// TwinCAT 3 PLC project Untitled1
// ProgramVersion: 3.1.4023.0
// libraries:
//   Tc2_Standard, * (Beckhoff Automation GmbH)
//   Tc2_System, * (Beckhoff Automation GmbH)
//   Tc2_TcpIp, * (Beckhoff Automation GmbH)
//   Tc3_Module, * (Beckhoff Automation GmbH)
//   Tc2_Utilities,3.3.47.0,Beckhoff Automation GmbH
//   VisuSymbols,3.5.10.0,System
// project tree:
//   / GlobalTextList.TcGTLO, PlcTask.TcTTO, Visualization Manager.TcVMO (not stored)
//   GVLs/ GVL.TcGVL
//   POUs/ MAIN.TcPOU
//   VISUs/ Visualization.TcVIS
// real-time tasks:
//   TASK PlcTask: cycle T#10ms, priority 20, ADS port 350

CONFIGURATION Untitled1
    RESOURCE PLC ON TwinCAT3
        TASK PlcTask(INTERVAL := T#10ms, PRIORITY := 20);
        PROGRAM MAIN WITH PlcTask : MAIN;
    END_RESOURCE
END_CONFIGURATION

// ---- GVLs/GVL.TcGVL
{attribute 'qualified_only'}
VAR_GLOBAL
	
	g_bStart    AT %I* : BOOL;
	g_nConnected : INT;
	g_sWinner : STRING;
	
	g_nShake1      : INT;
	g_nShake2    : INT;
	g_nShakeWin 				:INT := 500;
END_VAR

// ---- POUs/MAIN.TcPOU
PROGRAM MAIN
VAR
	fbUdpCreate 			: FB_SocketUdpCreate;
	fbUdpCreate2 			: FB_SocketUdpCreate;
	fbSocketSend  			: FB_SocketUdpSendTo;
	fbSocketReceive 		: FB_SocketUdpReceiveFrom;
	fbSocketSend2  			: FB_SocketUdpSendTo;
	fbSocketReceive2 		: FB_SocketUdpReceiveFrom;
	fbSocketClose			: FB_SocketClose;
	fbCloseAll				: FB_SocketCloseAll;	

	sLocalHost				: T_IPv4Addr 	:= '192.168.0.253';(* Local address: String containing an (Ipv4) Internet Protocol dotted address. *)
	nLocalPort				: UDINT			:= 24042;(* Local address: IP port number. *)
	nLocalPort2				: UDINT			:= 24043;(* Local address: IP port number. *)
	sRemoteHost				: T_IPv4Addr;// 	:= '192.168.0.101';(* Remote address: String containing an (Ipv4) Internet Protocol dotted address. *)
	nRemotePort				: UDINT 	;//	:= 62510;(* Remote address: IP port number. *)
	sRemoteHost2			: T_IPv4Addr;	(* Remote address: String containing an (Ipv4) Internet Protocol dotted address. *)
	nRemotePort2			: UDINT 	;   (* Remote address: IP port number. *)
	
	sOK						: STRING		:= 'B';
	sWIN					: STRING		:= 'W';
	sLOSE					: STRING		:= 'L';
	sNumberReceive			: STRING    	:= '';
	sNumberReceive2			: STRING    	:= '';
	sStartSignal			: STRING   		:= 'A';
	sStart					: STRING 		:= 'S';
	bInitialize				: BOOL := TRUE;
	bUdpCreated				: BOOL;
	bUdpCreated2			: BOOL;
	nState 					: INT;
	bEnable 				: BOOL 	:= TRUE;
	nErrorId    : UDINT;
	fbCreateTimer	: TON := ( PT := T#100MS);

	bVar					: BOOL;
	
	nShake1 				:INT := 0;
	nShake2 				:INT := 0;
	nNumber 				:INT := 0;
	pCurrentSocket 			:T_HSOCKET;
	hSocket: INT;
	nsh: BOOL;
END_VAR

fbCloseAll( bExecute:= bInitialize);
IF fbCloseAll.bBusy OR fbCloseAll.bError THEN
	nErrorId := fbCloseAll.nErrId;
	RETURN;
END_IF
bInitialize := FALSE;

//fbUdpCreate(nLocalPort := nLocalPort, sLocalHost := sLocalHost, bExecute := TRUE );

//fbSocketSend(nRemotePort := nRemotePort,  sRemoteHost := sRemoteHost, hSocket := fbUdpCreate.hSocket, cbLen := SIZEOF(nNumber), pSrc := ADR(nNumber), bExecute := TRUE);


CASE nState OF
0:
	IF bEnable THEN
		bUdpCreated := FALSE;
		nState := 1;
	END_IF
1:
	fbUdpCreate( bExecute := FALSE );
	fbUdpCreate2( bExecute := FALSE );
	fbUdpCreate( nLocalPort := nLocalPort, sLocalHost := sLocalHost, bExecute := TRUE );
	fbUdpCreate2( nLocalPort := nLocalPort2, sLocalHost := sLocalHost, bExecute := TRUE );
	nState := 2;
2:
	fbUdpCreate( bExecute:=FALSE );
	fbUdpCreate2( bExecute:=FALSE );
	IF NOT (fbUdpCreate.bBusy AND fbUdpCreate2.bBusy) THEN
		IF NOT (fbUdpCreate.bError AND fbUdpCreate2.bError) THEN
			bUdpCreated := TRUE;
			bUdpCreated2 := TRUE;
			//fbSocketReceive( bExecute := FALSE );
			
			fbSocketReceive( hSocket := fbUdpCreate.hSocket, cbLen := 1, pDest := ADR(sNumberReceive), bExecute := TRUE , tTimeout := T#100S);
			
			
			nState := 3;
		ELSE
			nState := 100;
		END_IF
	END_IF
3:

	fbSocketReceive( bExecute := FALSE );
		IF NOT fbSocketReceive.bBusy THEN
			IF NOT fbSocketReceive.bError THEN
				//nStringInt := StringToInt(in := sNumberReceive);
				IF (bVar := sNumberReceive <> 'A') THEN
					nState := 11;
				ELSE
					sRemoteHost := fbSocketReceive.sRemoteHost;
					nRemotePort := fbSocketReceive.nRemotePort;
					nState := 23;
					GVL.g_nConnected := 1;
					fbSocketReceive2( hSocket := fbUdpCreate2.hSocket, cbLen := 1, pDest := ADR(sNumberReceive2), bExecute := TRUE , tTimeout := T#100S);
				END_IF
				
			ELSE
				nState := 100;
			END_IF
		END_IF
23:
	fbSocketReceive2( bExecute := FALSE );
		IF NOT fbSocketReceive2.bBusy THEN
			IF NOT fbSocketReceive2.bError THEN
				//nStringInt := StringToInt(in := sNumberReceive);
				IF (bVar := sNumberReceive2 <> 'A') THEN
					nState := 211;
				ELSE
					sRemoteHost2 := fbSocketReceive2.sRemoteHost;
					nRemotePort2 := fbSocketReceive2.nRemotePort;
					nState := 40;
					GVL.g_nConnected := 2;
				END_IF
				
			ELSE
				nState := 100;
			END_IF
		END_IF	
//send S To Start game		
40:	
	fbSocketReceive( bExecute := FALSE );
	fbSocketReceive2( bExecute := FALSE );
	IF NOT fbSocketReceive.bBusy THEN
		fbSocketReceive( hSocket := fbUdpCreate.hSocket, cbLen := 1, pDest := ADR(sNumberReceive), bExecute := TRUE , tTimeout := T#10S);
	END_IF
	IF NOT fbSocketReceive2.bBusy THEN
		fbSocketReceive2( hSocket := fbUdpCreate2.hSocket, cbLen := 1, pDest := ADR(sNumberReceive2), bExecute := TRUE , tTimeout := T#10S);
	END_IF
	fbSocketSend( bExecute := FALSE );
	fbSocketSend2( bExecute := FALSE );
	IF NOT (fbSocketSend.bBusy AND fbSocketSend2.bBusy) THEN
		IF NOT (fbSocketSend.bError AND fbSocketSend2.bError) THEN	
			IF GVL.g_bStart THEN
			GVL.g_sWinner := '';
				GVL.g_nShake1 := 0;
				GVL.g_nShake2 := 0;
				sNumberReceive := '';
				sNumberReceive2 := '';
				//nCounterOut := nCounterOut + 1;
				fbSocketSend( bExecute := FALSE );
				fbSocketSend( nRemotePort := nRemotePort, sRemoteHost := sRemoteHost, hSocket := fbUdpCreate.hSocket, cbLen := 1, pSrc := ADR(sStart), bExecute := TRUE );
				fbSocketSend2( bExecute := FALSE );
				fbSocketSend2( nRemotePort := nRemotePort2, sRemoteHost := sRemoteHost2, hSocket := fbUdpCreate2.hSocket, cbLen := 1, pSrc := ADR(sStart), bExecute := TRUE );
				nState := 41;
			END_IF	
		END_IF
	END_IF
41:
	fbSocketSend( bExecute := FALSE );
	fbSocketSend2( bExecute := FALSE );
	IF NOT (fbSocketSend.bBusy AND fbSocketSend2.bBusy) THEN
		IF NOT (fbSocketSend.bError AND fbSocketSend2.bError) THEN
			
			nState := 4;
		ELSE
			nState := 100;
		END_IF
	END_IF
	
//send B To get values
4:

		//nCounterOut := nCounterOut + 1;
		fbSocketSend( bExecute := FALSE );
		fbSocketSend( nRemotePort := nRemotePort, sRemoteHost := sRemoteHost, hSocket := fbUdpCreate.hSocket, cbLen := 1, pSrc := ADR(sOK), bExecute := TRUE );
		fbSocketSend2( bExecute := FALSE );
		fbSocketSend2( nRemotePort := nRemotePort2, sRemoteHost := sRemoteHost2, hSocket := fbUdpCreate2.hSocket, cbLen := 1, pSrc := ADR(sOK), bExecute := TRUE );
		nState := 5;

5:
	fbSocketSend( bExecute := FALSE );
	fbSocketSend2( bExecute := FALSE );
	IF NOT (fbSocketSend.bBusy AND fbSocketSend2.bBusy) THEN
		IF NOT (fbSocketSend.bError AND fbSocketSend2.bError) THEN
			//fbSocketReceive( bExecute := FALSE );
			sNumberReceive := '';
			fbSocketReceive( hSocket := fbUdpCreate.hSocket, cbLen := 10, pDest := ADR(sNumberReceive), bExecute := TRUE , tTimeout := T#10S);
			sNumberReceive2 := '';
			fbSocketReceive2( hSocket := fbUdpCreate2.hSocket, cbLen := 10, pDest := ADR(sNumberReceive2), bExecute := TRUE , tTimeout := T#10S);
			nState := 6;
		ELSE
 			nState := 100;
		END_IF
	END_IF

//receive value
6:	
	fbSocketReceive( bExecute := FALSE );
	IF NOT fbSocketReceive.bBusy THEN
		IF NOT fbSocketReceive.bError THEN
		
			//fbSocketReceive( bExecute := FALSE );	
			IF (bVar := sNumberReceive = '') THEN
					nState := 4;
			END_IF
			
			IF(bVar := sNumberReceive = 'A') THEN
				sNumberReceive := '';
				fbSocketReceive( hSocket := fbUdpCreate.hSocket, cbLen := 10, pDest := ADR(sNumberReceive), bExecute := TRUE , tTimeout := T#10S);

			ELSE
					GVL.g_nShake1:= STRING_TO_WORD(sNumberReceive);
					nState := 26;

			END_IF
			
		ELSE
			nState := 100;
		END_IF
	END_IF
	
26:	
	fbSocketReceive2( bExecute := FALSE );
	IF NOT fbSocketReceive2.bBusy THEN
		IF NOT fbSocketReceive2.bError THEN
		
			//fbSocketReceive( bExecute := FALSE );	
			IF (bVar := sNumberReceive2 = '') THEN
					nState := 4;
			END_IF
			IF (bVar := sNumberReceive2 = 'A'	) THEN	
					
				sNumberReceive2 := '';
				fbSocketReceive2( hSocket := fbUdpCreate2.hSocket, cbLen := 10, pDest := ADR(sNumberReceive2), bExecute := TRUE , tTimeout := T#10S);

			ELSE
					GVL.g_nShake2:= STRING_TO_WORD(sNumberReceive2);
					nNumber := GVL.g_nShake1-GVL.g_nShake2;
					nState := 10;
					
					IF ( nNumber >= GVL.g_nShakeWin) THEN
						
						fbSocketSend( nRemotePort := nRemotePort, sRemoteHost := sRemoteHost, hSocket := fbUdpCreate.hSocket, cbLen := 1, pSrc := ADR(sWIN), bExecute := TRUE );
						fbSocketSend2( nRemotePort := nRemotePort2, sRemoteHost := sRemoteHost2, hSocket := fbUdpCreate2.hSocket, cbLen := 1, pSrc := ADR(sLOSE), bExecute := TRUE );
						nState := 40;
						GVL.g_sWinner := 'PLAYER 1 WON';
					END_IF
					
					IF ( nNumber <= -GVL.g_nShakeWin) THEN
						
						fbSocketSend( nRemotePort := nRemotePort, sRemoteHost := sRemoteHost, hSocket := fbUdpCreate.hSocket, cbLen := 1, pSrc := ADR(sLOSE), bExecute := TRUE );
						fbSocketSend2( nRemotePort := nRemotePort2, sRemoteHost := sRemoteHost2, hSocket := fbUdpCreate2.hSocket, cbLen := 1, pSrc := ADR(sWIN), bExecute := TRUE );
						nState := 40;
						GVL.g_sWinner := 'PLAYER 2 WON';
					END_IF
					
			END_IF

		ELSE
			nState := 100;
		END_IF
	END_IF
	
	
	
//timer and start after
10:
	fbCreateTimer( IN := TRUE);
	IF fbCreateTimer.Q THEN
		fbCreateTimer( IN := FALSE);
		nState := 4;
	END_IF
	//fbSocketDropMulticast( bExecute := FALSE );
	//fbSocketDropMulticast( hSocket := fbUdpCreate.hSocket, sMulticastAddr := sMulticastAddr, bExecute := TRUE );
//receive A
11:

	fbSocketReceive( hSocket := fbUdpCreate.hSocket, cbLen := 10, pDest := ADR(sNumberReceive), bExecute := TRUE , tTimeout := T#10S);
	nState := 3;
//receive message
211:

	fbSocketReceive2( hSocket := fbUdpCreate2.hSocket, cbLen := 10, pDest := ADR(sNumberReceive2), bExecute := TRUE , tTimeout := T#10S);
	nState := 23;
//receive message
12:

	fbSocketReceive( hSocket := fbUdpCreate.hSocket, cbLen := 10, pDest := ADR(sNumberReceive), bExecute := TRUE , tTimeout := T#10S);
	nState := 6;
	
//if disconnected or error
20:	
	fbSocketClose( bExecute := FALSE );
	fbSocketClose( hSocket := fbUdpCreate.hSocket, bExecute := TRUE );
	nState := 21;
21:	
	fbSocketClose( bExecute := FALSE );
	IF NOT fbSocketClose.bBusy THEN
		bUdpCreated := FALSE;
		IF NOT fbSocketClose.bError THEN
			nState := 0;	
		ELSE
			nState := 100;	
		END_IF
	END_IF
	
100:
	IF bUdpCreated THEN
		nState := 20;
	ELSE
		nState := 0;
	END_IF

END_CASE

END_PROGRAM

// ---- GlobalTextList.TcGTLO
TEXTLIST GlobalTextList
  915 = '"%d"'
  219 = '%d'
  938 = '%s'
  84 = 'PLAYER 1'
  796 = 'PLAYER 2'
  842 = 'players connected'
END_TEXTLIST

// ---- VISUs/Visualization.TcVIS
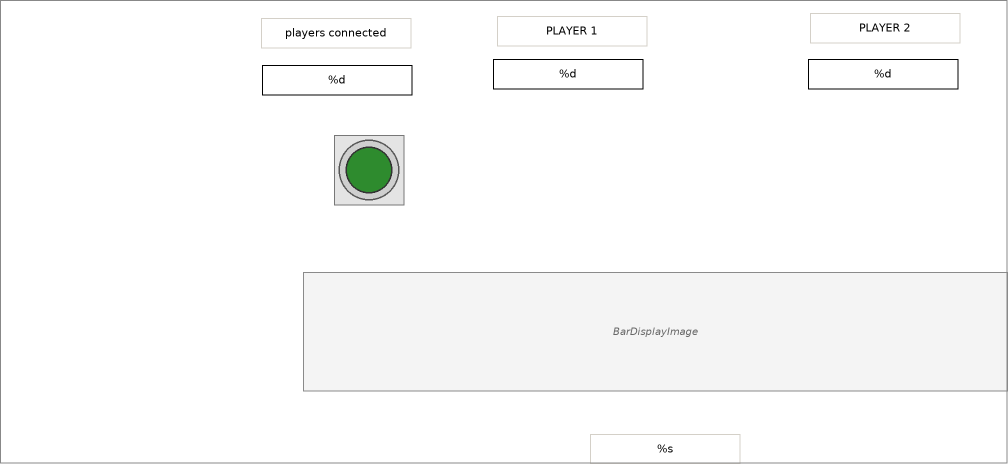
VISUALIZATION Visualization  // 1008x464
    PushSwitch (334,135 70x70), variable: GVL.g_bStart, behaviour: TAP, style: Switch-PushSwitch-Green
    Rectangle (493,59 150x30), "%d", text variable: GVL.g_nShake1
    Rectangle (808,59 150x30), "%d", text variable: GVL.g_nShake2
    Textfield (497,16 150x30), "PLAYER 1"
    Textfield (810,13 150x30), "PLAYER 2"
    Rectangle (262,65 150x30), "%d", text variable: GVL.g_nConnected
    Textfield (261,18 150x30), "players connected"
    Textfield (590,434 150x30), "%s", text variable: GVL.g_sWinner
    BarDisplayImage (303,272 705x119), value: GVL.g_nShake1-GVL.g_nShake2, style: BarDisplayImage-Gray, scale format: %.1f, scale -500..500
END_VISUALIZATION
